// TIA Portal V16 export
// export: Created 2021-11-12T13:32:45.3695002Z, ExportSetting WithDefaults, DisplayName Totally Integrated Automation Portal, DisplayVersion V16 Update 3, DisplayName TIA Portal Version Control Interface, DisplayVersion V16 Update 2, DisplayName TIA Portal Openness, DisplayVersion V16 Update 3, DisplayName SINAMICS Startdrive Advanced, DisplayVersion V16 Update 5, DisplayName SINAMICS Startdrive G130, G150, S120, S150, SINAMICS MV, S210, DisplayVersion V16 Update 5, DisplayName SINAMICS Startdrive G110M, G120, G120C, G120D, G120P, G115D, DisplayVersion V16 Update 5, DisplayName STEP 7 Professional, DisplayVersion V16 Update 3, DisplayName STEP 7 Safety, DisplayVersion V16, DisplayName WinCC UA Professional, DisplayVersion V16 Update 3
DATA_BLOCK "STATUS_BSN3"   // DB145
{ S7_Optimized_Access := 'TRUE' }
VERSION : 0.1
// stored: AutoNumber true, DBAccessibleFromOPCUA true, IsOnlyStoredInLoadMemory false, IsRetainMemResEnabled false, IsWriteProtectedInAS false, MemoryReserve 100
   VAR
      xxxxx___BinarySensors___xxxxx : Byte;
      xxxxx___BinaryOthers___xxxxx : Byte;
      xxxxx___AnalogueSensors___xxxxx : Byte;
      xxxxx___Drives___xxxxx : Byte;
      xxxxx___Other___xxxxx : Byte;
      Device : Struct   // Status of furnace
         Specific : "UDT_BSN3_Status_specific";
      END_STRUCT;
      "Counter" : Int;   // Number of parts in furnace
      CL01 : Struct   // Box for NOK parts / Bedna na NOK kusy
         Main : "UDT_Status_main";
         Specific { S7_SetPoint := 'True'} : "UDT_PartCounter_Status";
         Error { S7_SetPoint := 'True'} : "UDT_Error01";
      END_STRUCT;
      xxxxx___MaterialFlow___xxxxx : Byte;
      xxxxx__Alarms___xxxxx : Byte;
      Furnace : Struct   // From furnace / Sumární chyba z pece.
         Main : "UDT_Status_main";
         Specific : "UDT_DI_Mon_Status_specific";
         Error { S7_SetPoint := 'True'} : "UDT_Error01";
      END_STRUCT;
      LiveBit : Struct   // Communication / Chyba komunikace.
         Main : "UDT_Status_main";
         Specific : "UDT_DI_Mon_Status_specific";
         Error { S7_SetPoint := 'True'} : "UDT_Error01";
      END_STRUCT;
      DataTracking : Struct   // Part on senzor is not in data tracking / Kus na senzoru není na mapě.
         Main : "UDT_Status_main";
         Specific : "UDT_DI_Mon_Status_specific";
         Error { S7_SetPoint := 'True'} : "UDT_Error01";
      END_STRUCT;
      Senzor : Struct   // Part in data tracking is not on senzor / Kus na mapě není na senzoru.
         Main : "UDT_Status_main";
         Specific : "UDT_DI_Mon_Status_specific";
         Error { S7_SetPoint := 'True'} : "UDT_Error01";
      END_STRUCT;
      Alarm_5 : Struct
         Main : "UDT_Status_main";
         Specific : "UDT_DI_Mon_Status_specific";
         Error { S7_SetPoint := 'True'} : "UDT_Error01";
      END_STRUCT;
      Alarm_6 : Struct
         Main : "UDT_Status_main";
         Specific : "UDT_DI_Mon_Status_specific";
         Error { S7_SetPoint := 'True'} : "UDT_Error01";
      END_STRUCT;
      Alarm_7 : Struct
         Main : "UDT_Status_main";
         Specific : "UDT_DI_Mon_Status_specific";
         Error { S7_SetPoint := 'True'} : "UDT_Error01";
      END_STRUCT;
      Alarm_8 : Struct
         Main : "UDT_Status_main";
         Specific : "UDT_DI_Mon_Status_specific";
         Error { S7_SetPoint := 'True'} : "UDT_Error01";
      END_STRUCT;
      xxxxx___ProcessAlarms___xxxxx : Byte;
      CL01_Warn : Struct   // Box full warning / Varování plná bedna na kusy.
         Main : "UDT_Status_main";
         Specific { S7_SetPoint := 'True'} : "UDT_DI_Mon_Status_specific";
         Error { S7_SetPoint := 'True'} : "UDT_Error01";
      END_STRUCT;
      CL01_Alarm : Struct   // Box full alarm / Alarm plná bedna na kusy.
         Main : "UDT_Status_main";
         Specific : "UDT_DI_Mon_Status_specific";
         Error : "UDT_Error01";
      END_STRUCT;
      xxxxx__SafetyAlarms__xxxxx : Byte;
      ES : Struct   // Estop BSN3 / Estop BSN3.
         Main : "UDT_Status_main";
         Specific { S7_SetPoint := 'True'} : "UDT_DI_Mon_Status_specific";
         Error { S7_SetPoint := 'True'} : "UDT_Error01";
      END_STRUCT;
   END_VAR
BEGIN
END_DATA_BLOCK
